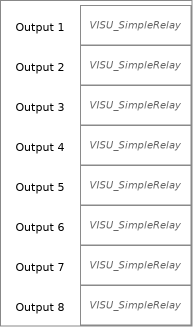
VISUALIZATION VISU_TelemetryFlatfieldLeds  // 193x327
VAR_IN_OUT
	ref : TelemetryFlatfieldLeds;
    widget : TelemetryFlatfieldLedsWidget;
END_VAR
    Frame (80,5 111x40)
        shows VISU_SimpleRelay(ref := ref.parts.output1, widget := widget.output1)
    Label (5,10 70x35), "Output 1"
    Frame (80,45 111x40)
        shows VISU_SimpleRelay(ref := ref.parts.output2, widget := widget.output2)
    Label (5,50 70x35), "Output 2"
    Frame (80,85 111x40)
        shows VISU_SimpleRelay(ref := ref.parts.output3, widget := widget.output3)
    Label (5,90 70x35), "Output 3"
    Frame (80,125 111x40)
        shows VISU_SimpleRelay(ref := ref.parts.output4, widget := widget.output4)
    Label (5,130 70x35), "Output 4"
    Frame (80,165 111x40)
        shows VISU_SimpleRelay(ref := ref.parts.output5, widget := widget.output5)
    Label (5,170 70x35), "Output 5"
    Frame (80,205 111x40)
        shows VISU_SimpleRelay(ref := ref.parts.output6, widget := widget.output6)
    Label (5,210 70x35), "Output 6"
    Frame (80,245 111x40)
        shows VISU_SimpleRelay(ref := ref.parts.output7, widget := widget.output7)
    Label (5,250 70x35), "Output 7"
    Frame (80,285 111x40)
        shows VISU_SimpleRelay(ref := ref.parts.output8, widget := widget.output8)
    Label (5,290 70x35), "Output 8"
END_VISUALIZATION

(* stored: Version 1.1.0.1, ProductVersion 3.1.4019.2
   Visu VISU_TelemetryFlatfieldLeds: Id {2b1921e1-93b7-4f22-a690-67197b28699d} *)
